(* CODESYS project LadderAndST.project

Project tree, tasks and I/O mapping:
  Device : CODESYS Control Win V3, 3S - Smart Software Solutions GmbH, order no. 305021, version 3.5.10.30
    application Application
      libraries: Standard, * (System)
      task MainTask (cyclic, interval t#20ms, priority 1) calls PLC_PRG, ST_PRG
      task VISU_TASK (cyclic, interval 100 ms, priority 31) calls VisuElems.Visu_Prg
      program PLC_PRG [LD]
      visualisation Visualization1
      program ST_PRG [ST]
  libraries: VisuSymbols, 3.5.10.0 (System)
  text list GlobalTextList
*)

// Device/Application/PLC_PRG
PROGRAM PLC_PRG
VAR
	Contact1: BOOL := FALSE;
	Coil1: BOOL;
	Contact2: BOOL := FALSE;
	Contact3: BOOL := TRUE;
END_VAR

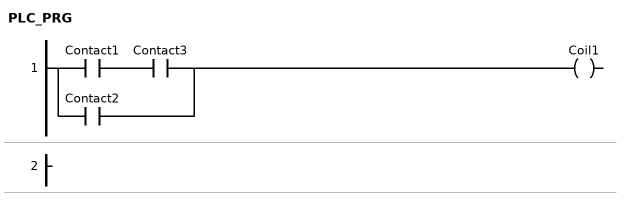
// NETWORK 1
Coil1 := Contact1 AND Contact3 OR Contact2;

// NETWORK 2

END_PROGRAM

// Device/Application/ST_PRG
PROGRAM ST_PRG
VAR
	Contact1: BOOL := FALSE ;
	Contact2: BOOL := FALSE;
	Contact3: BOOL := FALSE;
	Coil1: BOOL := FALSE ;
END_VAR

IF (Contact1 = TRUE AND contact2 = TRUE) OR contact3 = TRUE THEN;
	Coil1 := TRUE;
ELSE;
	Coil1 := FALSE; 
END_IF

END_PROGRAM

// Device/Application/Visualization1
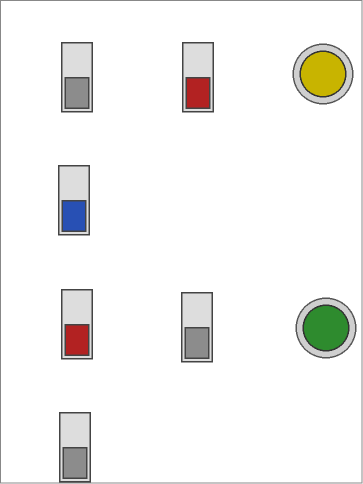
VISUALIZATION Visualization1  // 363x484
    DipSwitch (42,42 70x70), variable: PLC_PRG.Contact1, behaviour: TOGGLE, style: Switch-DipSwitch-Gray
    Lamp1 (288,39 70x70), variable: PLC_PRG.Coil1, style: Lamp-Lamp1-Yellow
    DipSwitch (39,165 70x70), variable: PLC_PRG.Contact2, behaviour: TOGGLE, style: Switch-DipSwitch-Blue
    DipSwitch (163,42 70x70), variable: PLC_PRG.Contact3, behaviour: TOGGLE, style: Switch-DipSwitch-Red
    Lamp1 (291,293 70x70), variable: ST_PRG.Coil1, style: Lamp-Lamp1-Green
    DipSwitch (42,289 70x70), variable: ST_PRG.Contact1, behaviour: TOGGLE, style: Switch-DipSwitch-Red
    DipSwitch (162,292 70x70), variable: ST_PRG.Contact2, behaviour: TOGGLE, style: Switch-DipSwitch-Gray
    DipSwitch (40,412 70x70), variable: ST_PRG.Contact3, behaviour: TOGGLE, style: Switch-DipSwitch-Gray
END_VISUALIZATION
